TYPE INTERNAL FrameMeta :
STRUCT
  {attribute 'displaymode':='hex'}
  Id : UDINT;
  Size : DINT;
  TotalDuration : LWORD; 
END_STRUCT
END_TYPE

(* stored: Version 1.1.0.1, ProductVersion 3.1.4024.9
   DUT FrameMeta: Id {be0a15a5-1190-4803-b2b2-e0863c074c6c} *)
